(* Logix 5000 project; controller Project_Template vendor 1 type 14 code 106 rev 33.12; software revision 33.00 *)

TASK MainTask (continuous, watchdog 500 ms) : MainProgram

MODULES
   Local : vendor 1 type 14 code 106 (Compact 0, rev 33.12)
      Discrete_In_Slot_3 : 1769-IQ16 (Compact 3, rev 1.1, Input RPI 20 ms)
      Discrete_In_Slot_2 : 1769-IQ16 (Compact 2, rev 1.1, Input RPI 20 ms)
      ASCII_Slot_1 : vendor 1 type 109 code 66 (Compact 1, rev 2.1, Output RPI 100 ms)
      Discrete_Out_Slot_4 : 1769-OW16 (Compact 4, rev 1.1, Output RPI 20 ms)
      Discrete_Out_Slot_5 : 1769-OW16 (Compact 5, rev 1.1, Output RPI 20 ms)
END_MODULES

VAR_GLOBAL   (* controller tags *)
   AT_HOME : BOOL := 1;   // Home position
   AUTO : BOOL;   // Set Auto Process
   Box_Fell : BOOL;
   FLASH_FAST : BOOL;
   Flash_Fast_Off : TIMER := (PRE := 250);
   Flash_Fast_On : TIMER := (PRE := 250, ACC := 161, EN := 1, TT := 1);
   FLASH_MEDIUM : BOOL := 1;
   Flash_Medium_Off : TIMER := (PRE := 500, ACC := 161, EN := 1, TT := 1);
   Flash_Medium_On : TIMER := (PRE := 500, ACC := 500, EN := 1, DN := 1);
   FLASH_SLOW : BOOL;   // Slow Flashing
   Flash_Slow_Off : TIMER := (PRE := 1000);
   Flash_Slow_On : TIMER := (PRE := 1000, ACC := 664, EN := 1, TT := 1);
   I_Auto_Mode_Selector : ALIAS FOR Local:2:I.Data.2;
   I_Barcode_Stop_Raised : ALIAS FOR Local:3:I.Data.1;
   I_Box_Ejector_Extended : ALIAS FOR Local:2:I.Data.4;
   I_Reject_Cyl_Lowered : ALIAS FOR Local:3:I.Data.2;
   I_Reset_PB : ALIAS FOR Local:2:I.Data.3;
   I_Start_PB : ALIAS FOR Local:2:I.Data.0;
   I_Stop_PB : ALIAS FOR Local:2:I.Data.1;
   I_Vacuum_Head_at_Conveyor : ALIAS FOR Local:3:I.Data.0;
   I_Vacuum_Head_at_Magazine : ALIAS FOR Local:2:I.Data.15;
   I_Vacuum_Head_Extended : ALIAS FOR Local:2:I.Data.14;
   I_Vacuum_Head_Lowered : ALIAS FOR Local:2:I.Data.10;
   I_Vacuum_Head_Raised : ALIAS FOR Local:2:I.Data.9;
   I_Vacuum_Head_Retracted : ALIAS FOR Local:2:I.Data.13;
   I_Vacuum_Head_Rotated_CCW : ALIAS FOR Local:2:I.Data.11;
   I_Vacuum_Head_Rotated_CW : ALIAS FOR Local:2:I.Data.12;
   I_Vacuum_Sensor_On : ALIAS FOR Local:3:I.Data.8;
   O_Amber_Tower_Ind : ALIAS FOR Local:5:O.Data.9;
   O_Barcode_Stop_Raise : ALIAS FOR Local:4:O.Data.14;
   O_Box_Eject : ALIAS FOR Local:4:O.Data.0;
   O_Conveyor_On : ALIAS FOR Local:5:O.Data.5;
   O_Green_Tower_Ind : ALIAS FOR Local:5:O.Data.8;
   O_Red_Tower_Ind : ALIAS FOR Local:5:O.Data.10;
   O_Reject_Cyl_Extend : ALIAS FOR Local:5:O.Data.0;
   O_Reject_Cyl_Lower : ALIAS FOR Local:4:O.Data.15;
   O_Vacuum_Head_Extend : ALIAS FOR Local:4:O.Data.8;
   O_Vacuum_Head_Lower : ALIAS FOR Local:4:O.Data.5;
   O_Vacuum_Head_Rotate_CCW : ALIAS FOR Local:4:O.Data.7;
   O_Vacuum_Head_Rotate_CW : ALIAS FOR Local:4:O.Data.6;
   O_Vacuum_Head_to_Conveyor : ALIAS FOR Local:4:O.Data.9;
   O_Vacuum_Head_to_Magazine : ALIAS FOR Local:4:O.Data.10;
   O_Vacuum_Off : ALIAS FOR Local:5:O.Data.2;
   O_Vacuum_On : ALIAS FOR Local:5:O.Data.1;
   Production_Step : DINT := 11;
   Raise_Vacuum : BOOL;
   Reset_Step : DINT := 512;
   Retract_Box_Ejector : BOOL;
   Retract_Vacuum : BOOL;
   Status_IN_PRODUCTION : BOOL;
   Status_RESETTING : BOOL;
   Timer_Barcode_Delay : TIMER := (PRE := 1000);
   Timer_Conveyor_Delay : TIMER := (PRE := 500);
   Timer_Conveyor_Reset : TIMER := (PRE := 900, ACC := 900, EN := 1, DN := 1);   // Timer Conveyor to clear boxes
   Timer_Extend_Delay : TIMER := (PRE := 2000, ACC := 296, EN := 1, TT := 1);
   Timer_Pre_Production : TIMER := (PRE := 500, ACC := 500, EN := 1, DN := 1);
   Timer_Pre_Reset : TIMER := (PRE := 500);
   Timer_Reset : TIMER[7] := ([0].PRE := 250, [1].PRE := 250, [2].PRE := 250, [3].PRE := 250, [4].PRE := 250, [5].PRE := 300, [6].PRE := 125);
   Timer_Vacuum_Delay : TIMER := (PRE := 250, ACC := 250, EN := 1, DN := 1);
END_VAR

PROGRAM MainProgram   (* main routine MainRoutine *)

ROUTINE a_Reset_Routine   (* ladder *)
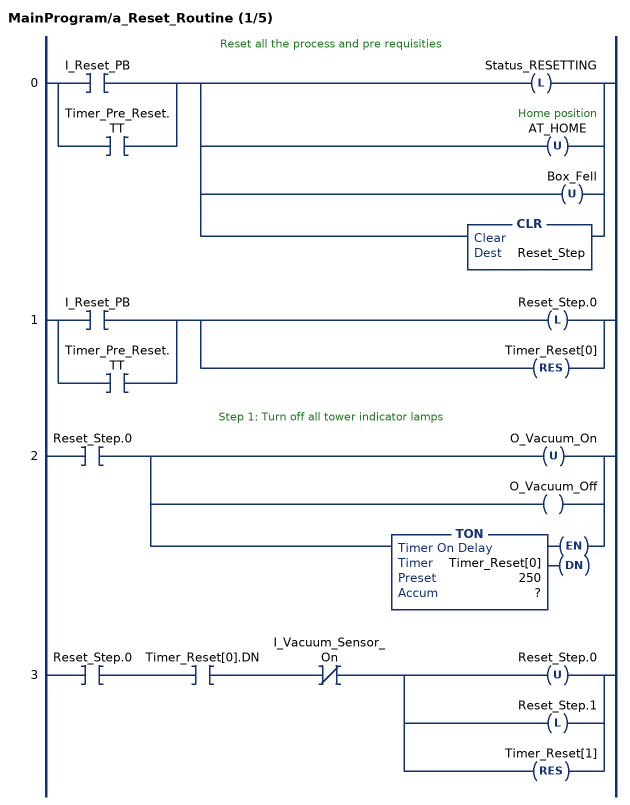
   // Reset all the process and pre requisities
   0: [XIC(I_Reset_PB) ,XIC(Timer_Pre_Reset.TT) ][OTL(Status_RESETTING) ,OTU(AT_HOME) ,OTU(Box_Fell) ,CLR(Reset_Step) ];
   1: [XIC(I_Reset_PB) ,XIC(Timer_Pre_Reset.TT) ][OTL(Reset_Step.0) ,RES(Timer_Reset[0]) ];
   // Step 1: Turn off all tower indicator lamps
   2: XIC(Reset_Step.0)[OTU(O_Vacuum_On) ,OTE(O_Vacuum_Off) ,TON(Timer_Reset[0],?,?) ];
   3: XIC(Reset_Step.0)XIC(Timer_Reset[0].DN)XIO(I_Vacuum_Sensor_On)[OTU(Reset_Step.0) ,OTL(Reset_Step.1) ,RES(Timer_Reset[1]) ];
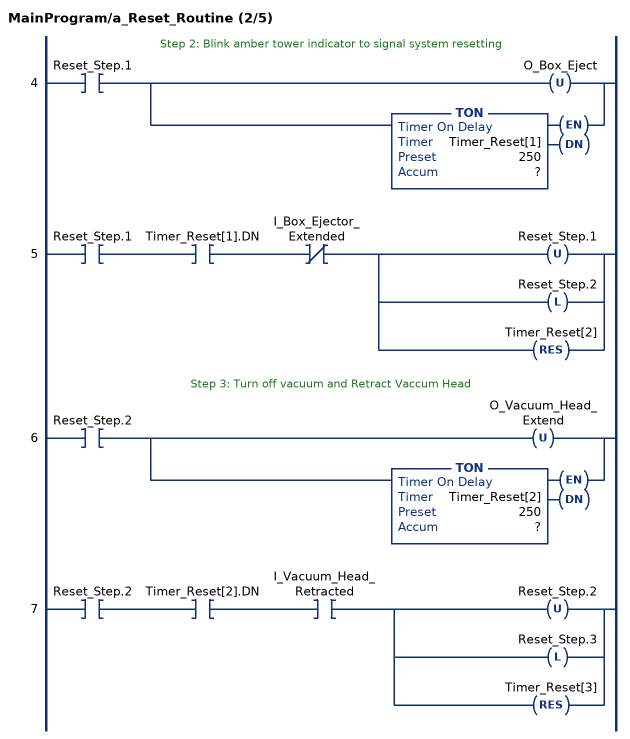
   // Step 2: Blink amber tower indicator to signal system resetting
   4: XIC(Reset_Step.1)[OTU(O_Box_Eject) ,TON(Timer_Reset[1],?,?) ];
   5: XIC(Reset_Step.1)XIC(Timer_Reset[1].DN)XIO(I_Box_Ejector_Extended)[OTU(Reset_Step.1) ,OTL(Reset_Step.2) ,RES(Timer_Reset[2]) ];
   // Step 3: Turn off vacuum and Retract Vaccum Head
   6: XIC(Reset_Step.2)[OTU(O_Vacuum_Head_Extend) ,TON(Timer_Reset[2],?,?) ];
   7: XIC(Reset_Step.2)XIC(Timer_Reset[2].DN)XIC(I_Vacuum_Head_Retracted)[OTU(Reset_Step.2) ,OTL(Reset_Step.3) ,RES(Timer_Reset[3]) ];
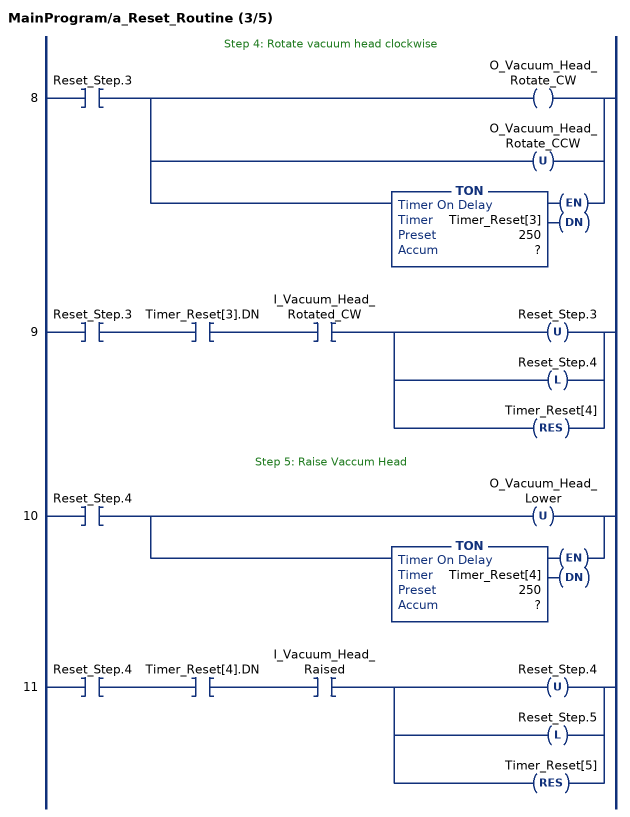
   // Step 4: Rotate vacuum head clockwise
   8: XIC(Reset_Step.3)[OTE(O_Vacuum_Head_Rotate_CW) ,OTU(O_Vacuum_Head_Rotate_CCW) ,TON(Timer_Reset[3],?,?) ];
   9: XIC(Reset_Step.3)XIC(Timer_Reset[3].DN)XIC(I_Vacuum_Head_Rotated_CW)[OTU(Reset_Step.3) ,OTL(Reset_Step.4) ,RES(Timer_Reset[4]) ];
   // Step 5: Raise Vaccum Head
   10: XIC(Reset_Step.4)[OTU(O_Vacuum_Head_Lower) ,TON(Timer_Reset[4],?,?) ];
   11: XIC(Reset_Step.4)XIC(Timer_Reset[4].DN)XIC(I_Vacuum_Head_Raised)[OTU(Reset_Step.4) ,OTL(Reset_Step.5) ,RES(Timer_Reset[5]) ];
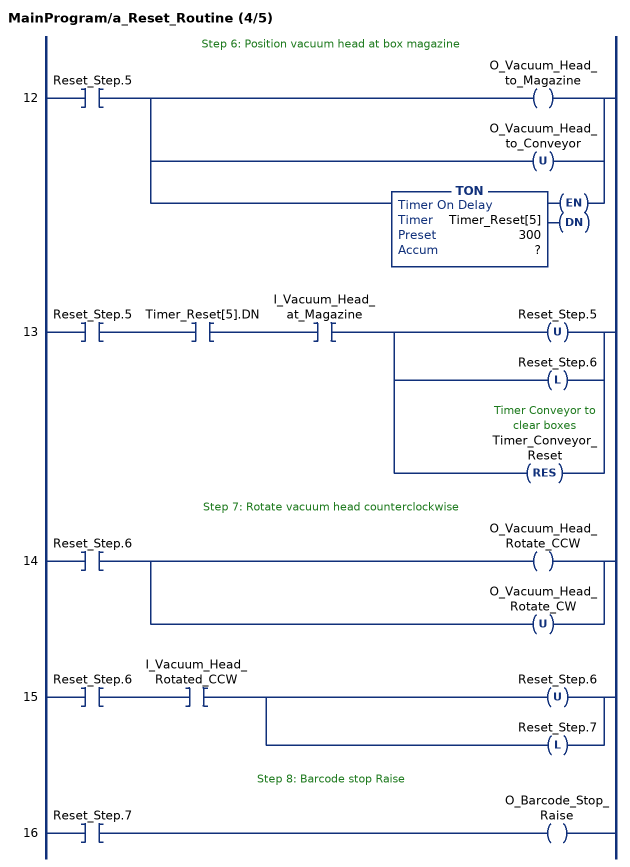
   // Step 6: Position vacuum head at box magazine
   12: XIC(Reset_Step.5)[OTE(O_Vacuum_Head_to_Magazine) ,OTU(O_Vacuum_Head_to_Conveyor) ,TON(Timer_Reset[5],?,?) ];
   13: XIC(Reset_Step.5)XIC(Timer_Reset[5].DN)XIC(I_Vacuum_Head_at_Magazine)[OTU(Reset_Step.5) ,OTL(Reset_Step.6) ,RES(Timer_Conveyor_Reset) ];
   // Step 7: Rotate vacuum head counterclockwise
   14: XIC(Reset_Step.6)[OTE(O_Vacuum_Head_Rotate_CCW) ,OTU(O_Vacuum_Head_Rotate_CW) ];
   15: XIC(Reset_Step.6)XIC(I_Vacuum_Head_Rotated_CCW)[OTU(Reset_Step.6) ,OTL(Reset_Step.7) ];
   // Step 8: Barcode stop Raise
   16: XIC(Reset_Step.7)OTE(O_Barcode_Stop_Raise);
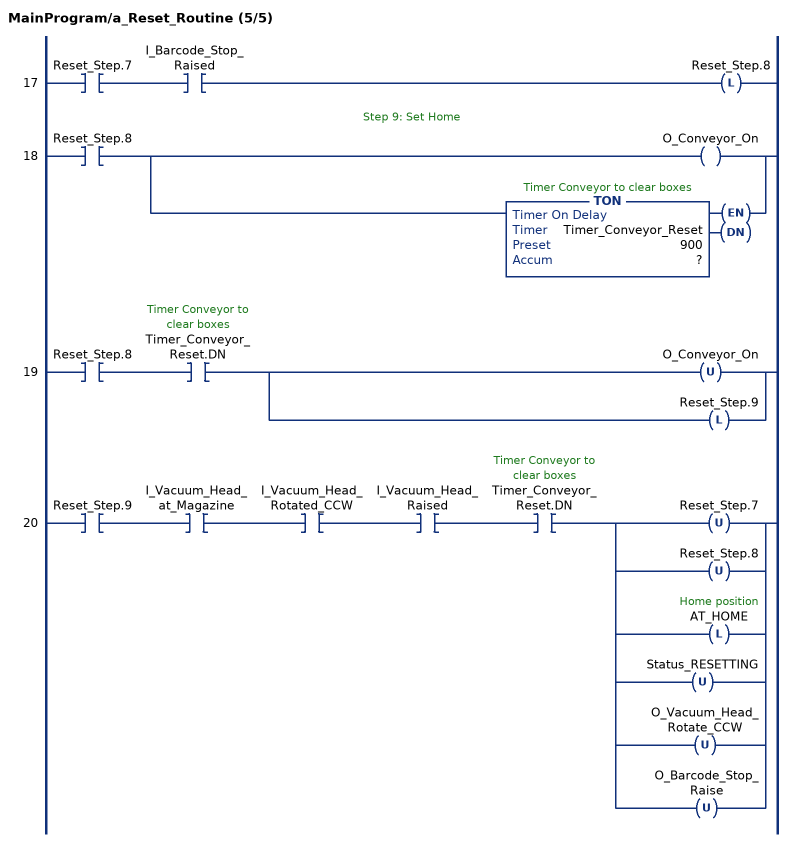
   17: XIC(Reset_Step.7)XIC(I_Barcode_Stop_Raised)OTL(Reset_Step.8);
   // Step 9: Set Home
   18: XIC(Reset_Step.8)[OTE(O_Conveyor_On) ,TON(Timer_Conveyor_Reset,?,?) ];
   19: XIC(Reset_Step.8)XIC(Timer_Conveyor_Reset.DN)[OTU(O_Conveyor_On) ,OTL(Reset_Step.9) ];
   20: XIC(Reset_Step.9)XIC(I_Vacuum_Head_at_Magazine)XIC(I_Vacuum_Head_Rotated_CCW)XIC(I_Vacuum_Head_Raised)XIC(Timer_Conveyor_Reset.DN)[OTU(Reset_Step.7) ,OTU(Reset_Step.8) ,OTL(AT_HOME) ,OTU(Status_RESETTING) ,OTU(O_Vacuum_Head_Rotate_CCW) ,OTU(O_Barcode_Stop_Raise) ];
END_ROUTINE

ROUTINE b_Production_Routine   (* ladder *)
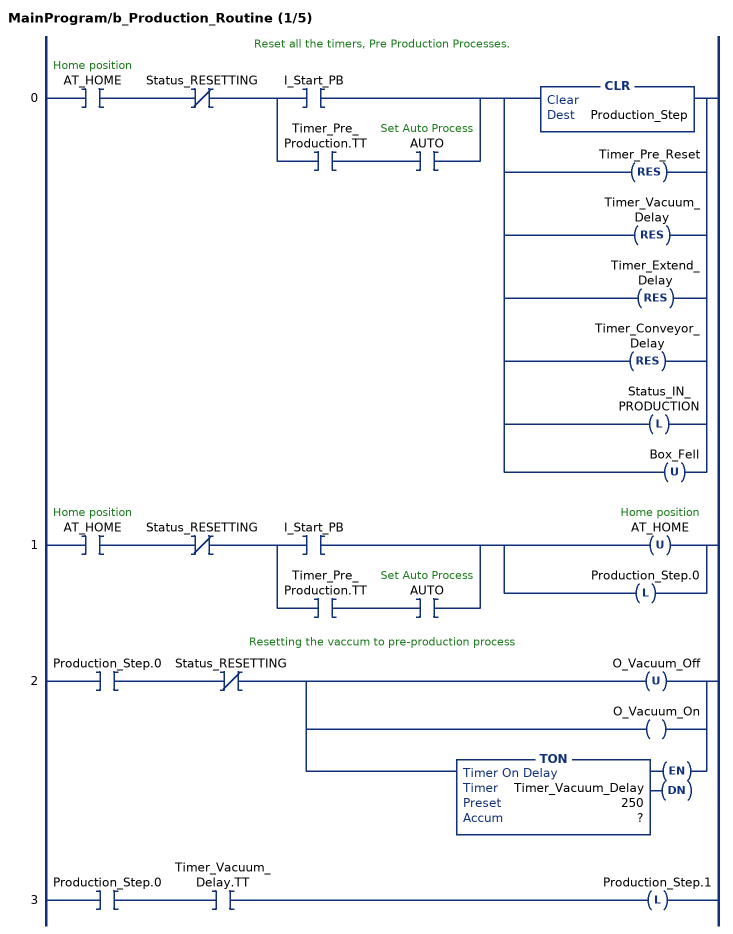
   // Reset all the timers, Pre Production Processes.
   0: XIC(AT_HOME)XIO(Status_RESETTING)[XIC(I_Start_PB) ,XIC(Timer_Pre_Production.TT) XIC(AUTO) ][CLR(Production_Step) ,RES(Timer_Pre_Reset) ,RES(Timer_Vacuum_Delay) ,RES(Timer_Extend_Delay) ,RES(Timer_Conveyor_Delay) ,OTL(Status_IN_PRODUCTION) ,OTU(Box_Fell) ];
   1: XIC(AT_HOME)XIO(Status_RESETTING)[XIC(I_Start_PB) ,XIC(Timer_Pre_Production.TT) XIC(AUTO) ][OTU(AT_HOME) ,OTL(Production_Step.0) ];
   // Resetting the vaccum to pre-production process
   2: XIC(Production_Step.0)XIO(Status_RESETTING)[OTU(O_Vacuum_Off) ,OTE(O_Vacuum_On) ,TON(Timer_Vacuum_Delay,?,?) ];
   3: XIC(Production_Step.0)XIC(Timer_Vacuum_Delay.TT)OTL(Production_Step.1);
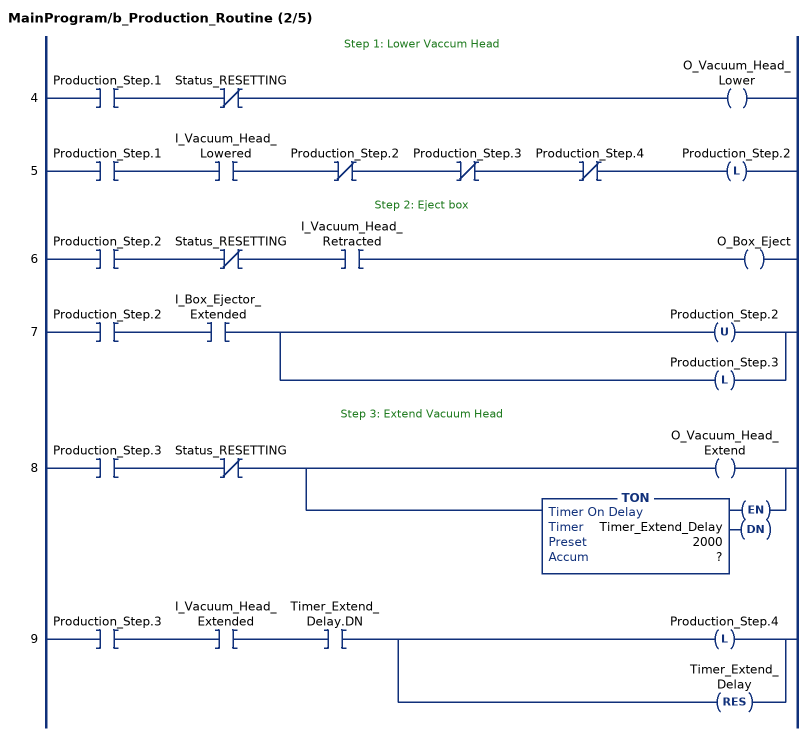
   // Step 1: Lower Vaccum Head
   4: XIC(Production_Step.1)XIO(Status_RESETTING)OTE(O_Vacuum_Head_Lower);
   5: XIC(Production_Step.1)XIC(I_Vacuum_Head_Lowered)XIO(Production_Step.2)XIO(Production_Step.3)XIO(Production_Step.4)OTL(Production_Step.2);
   // Step 2: Eject box
   6: XIC(Production_Step.2)XIO(Status_RESETTING)XIC(I_Vacuum_Head_Retracted)OTE(O_Box_Eject);
   7: XIC(Production_Step.2)XIC(I_Box_Ejector_Extended)[OTU(Production_Step.2) ,OTL(Production_Step.3) ];
   // Step 3: Extend Vacuum Head
   8: XIC(Production_Step.3)XIO(Status_RESETTING)[OTE(O_Vacuum_Head_Extend) ,TON(Timer_Extend_Delay,?,?) ];
   9: XIC(Production_Step.3)XIC(I_Vacuum_Head_Extended)XIC(Timer_Extend_Delay.DN)[OTL(Production_Step.4) ,RES(Timer_Extend_Delay) ];
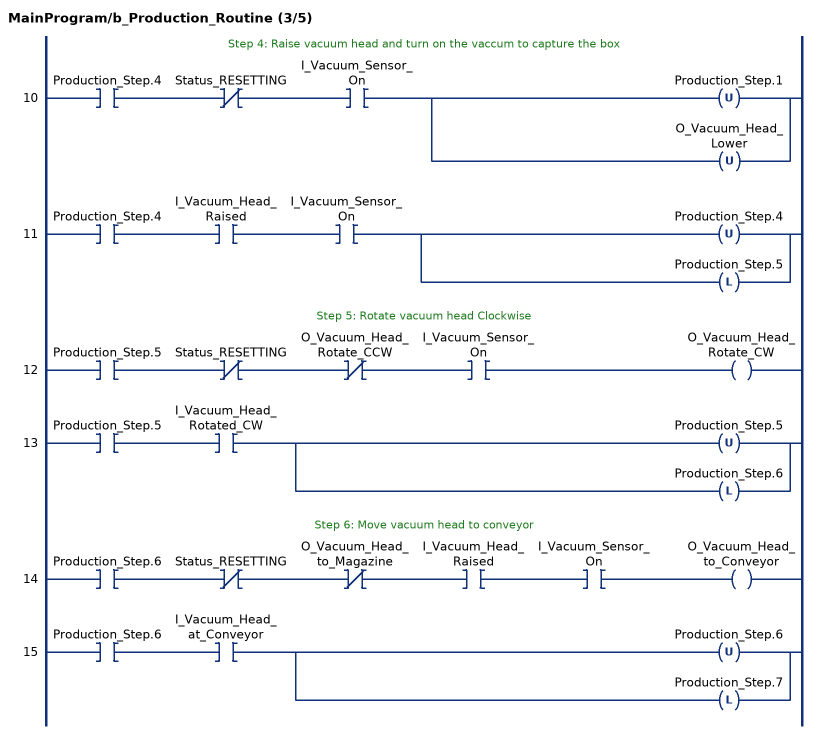
   // Step 4: Raise vacuum head and turn on the vaccum to capture the box
   10: XIC(Production_Step.4)XIO(Status_RESETTING)XIC(I_Vacuum_Sensor_On)[OTU(Production_Step.1) ,OTU(O_Vacuum_Head_Lower) ];
   11: XIC(Production_Step.4)XIC(I_Vacuum_Head_Raised)XIC(I_Vacuum_Sensor_On)[OTU(Production_Step.4) ,OTL(Production_Step.5) ];
   // Step 5: Rotate vacuum head Clockwise
   12: XIC(Production_Step.5)XIO(Status_RESETTING)XIO(O_Vacuum_Head_Rotate_CCW)XIC(I_Vacuum_Sensor_On)OTE(O_Vacuum_Head_Rotate_CW);
   13: XIC(Production_Step.5)XIC(I_Vacuum_Head_Rotated_CW)[OTU(Production_Step.5) ,OTL(Production_Step.6) ];
   // Step 6: Move vacuum head to conveyor
   14: XIC(Production_Step.6)XIO(Status_RESETTING)XIO(O_Vacuum_Head_to_Magazine)XIC(I_Vacuum_Head_Raised)XIC(I_Vacuum_Sensor_On)OTE(O_Vacuum_Head_to_Conveyor);
   15: XIC(Production_Step.6)XIC(I_Vacuum_Head_at_Conveyor)[OTU(Production_Step.6) ,OTL(Production_Step.7) ];
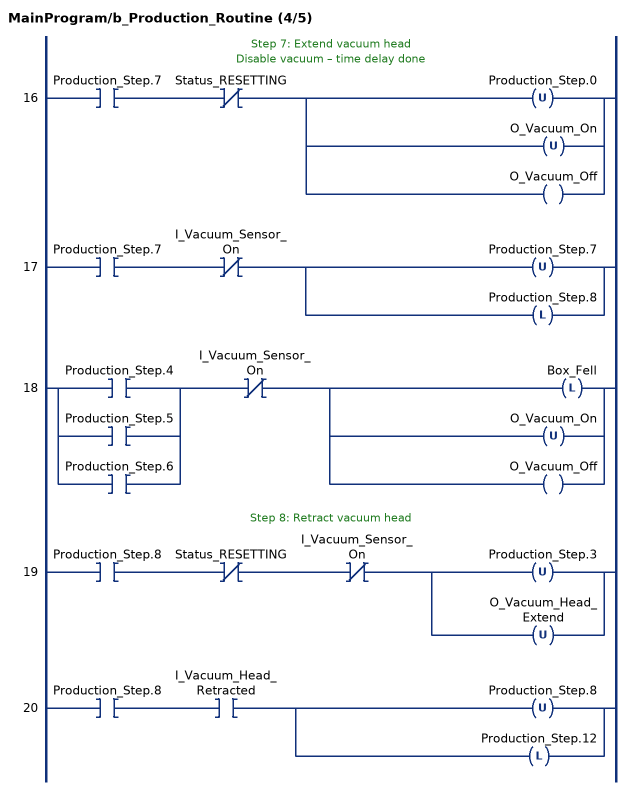
   // Step 7: Extend vacuum head
   // Disable vacuum – time delay done
   16: XIC(Production_Step.7)XIO(Status_RESETTING)[OTU(Production_Step.0) ,OTU(O_Vacuum_On) ,OTE(O_Vacuum_Off) ];
   17: XIC(Production_Step.7)XIO(I_Vacuum_Sensor_On)[OTU(Production_Step.7) ,OTL(Production_Step.8) ];
   18: [XIC(Production_Step.4) ,XIC(Production_Step.5) ,XIC(Production_Step.6) ]XIO(I_Vacuum_Sensor_On)[OTL(Box_Fell) ,OTU(O_Vacuum_On) ,OTE(O_Vacuum_Off) ];
   // Step 8: Retract vacuum head
   19: XIC(Production_Step.8)XIO(Status_RESETTING)XIO(I_Vacuum_Sensor_On)[OTU(Production_Step.3) ,OTU(O_Vacuum_Head_Extend) ];
   20: XIC(Production_Step.8)XIC(I_Vacuum_Head_Retracted)[OTU(Production_Step.8) ,OTL(Production_Step.12) ];
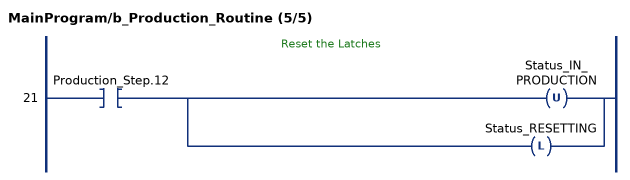
   // Reset the Latches
   21: XIC(Production_Step.12)[OTU(Status_IN_PRODUCTION) ,OTL(Status_RESETTING) ];
END_ROUTINE

ROUTINE c_AutoProcess_Routine   (* ladder *)
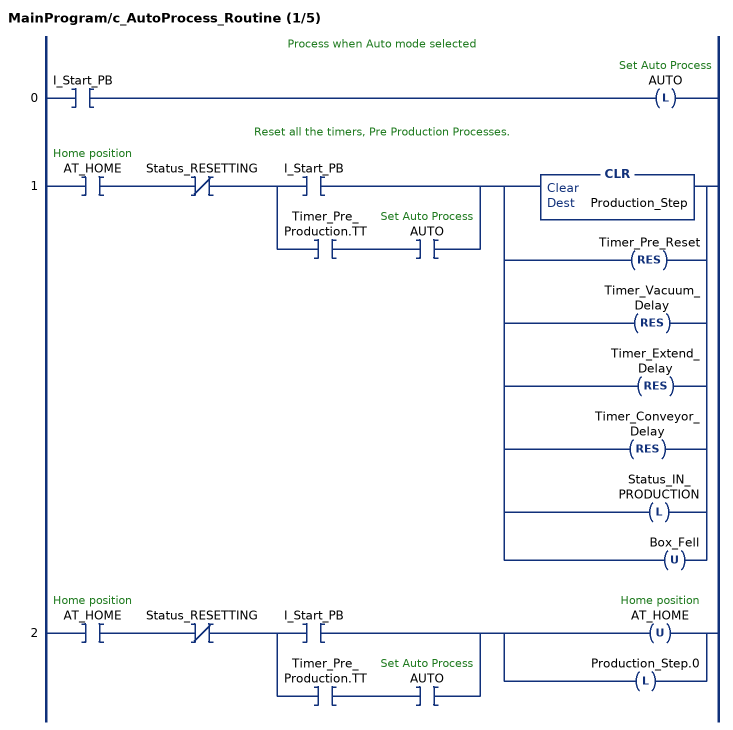
   // Process when Auto mode selected
   0: XIC(I_Start_PB)OTL(AUTO);
   // Reset all the timers, Pre Production Processes.
   1: XIC(AT_HOME)XIO(Status_RESETTING)[XIC(I_Start_PB) ,XIC(Timer_Pre_Production.TT) XIC(AUTO) ][CLR(Production_Step) ,RES(Timer_Pre_Reset) ,RES(Timer_Vacuum_Delay) ,RES(Timer_Extend_Delay) ,RES(Timer_Conveyor_Delay) ,OTL(Status_IN_PRODUCTION) ,OTU(Box_Fell) ];
   2: XIC(AT_HOME)XIO(Status_RESETTING)[XIC(I_Start_PB) ,XIC(Timer_Pre_Production.TT) XIC(AUTO) ][OTU(AT_HOME) ,OTL(Production_Step.0) ];
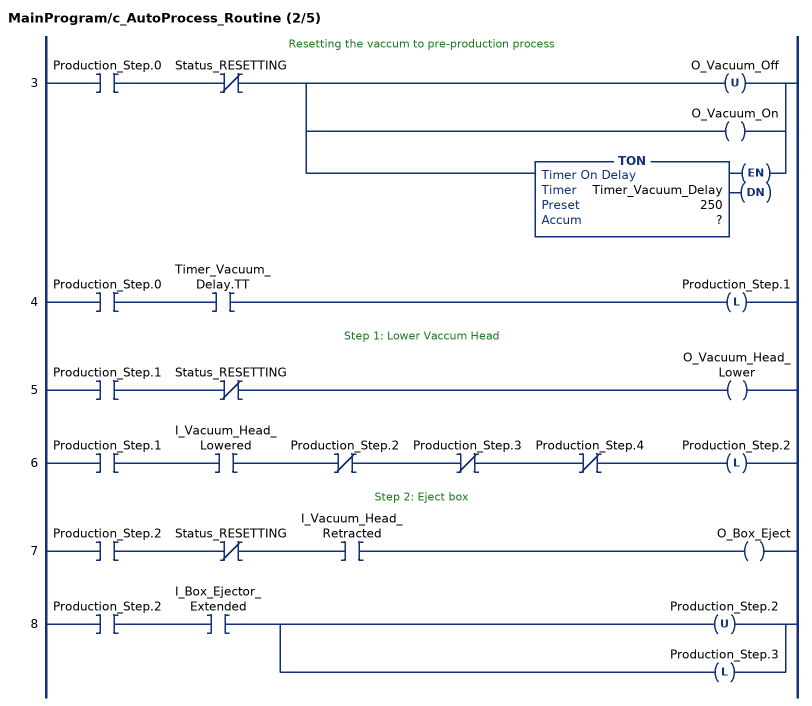
   // Resetting the vaccum to pre-production process
   3: XIC(Production_Step.0)XIO(Status_RESETTING)[OTU(O_Vacuum_Off) ,OTE(O_Vacuum_On) ,TON(Timer_Vacuum_Delay,?,?) ];
   4: XIC(Production_Step.0)XIC(Timer_Vacuum_Delay.TT)OTL(Production_Step.1);
   // Step 1: Lower Vaccum Head
   5: XIC(Production_Step.1)XIO(Status_RESETTING)OTE(O_Vacuum_Head_Lower);
   6: XIC(Production_Step.1)XIC(I_Vacuum_Head_Lowered)XIO(Production_Step.2)XIO(Production_Step.3)XIO(Production_Step.4)OTL(Production_Step.2);
   // Step 2: Eject box
   7: XIC(Production_Step.2)XIO(Status_RESETTING)XIC(I_Vacuum_Head_Retracted)OTE(O_Box_Eject);
   8: XIC(Production_Step.2)XIC(I_Box_Ejector_Extended)[OTU(Production_Step.2) ,OTL(Production_Step.3) ];
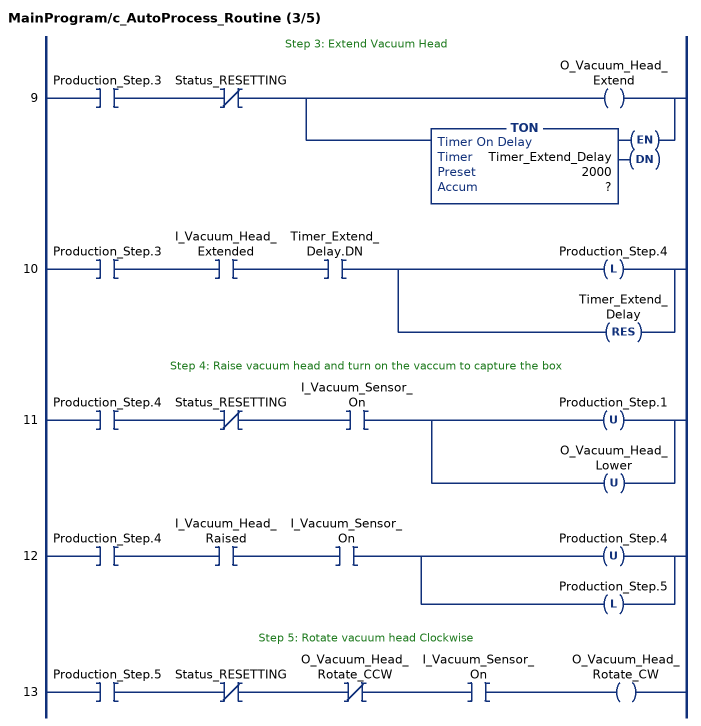
   // Step 3: Extend Vacuum Head
   9: XIC(Production_Step.3)XIO(Status_RESETTING)[OTE(O_Vacuum_Head_Extend) ,TON(Timer_Extend_Delay,?,?) ];
   10: XIC(Production_Step.3)XIC(I_Vacuum_Head_Extended)XIC(Timer_Extend_Delay.DN)[OTL(Production_Step.4) ,RES(Timer_Extend_Delay) ];
   // Step 4: Raise vacuum head and turn on the vaccum to capture the box
   11: XIC(Production_Step.4)XIO(Status_RESETTING)XIC(I_Vacuum_Sensor_On)[OTU(Production_Step.1) ,OTU(O_Vacuum_Head_Lower) ];
   12: XIC(Production_Step.4)XIC(I_Vacuum_Head_Raised)XIC(I_Vacuum_Sensor_On)[OTU(Production_Step.4) ,OTL(Production_Step.5) ];
   // Step 5: Rotate vacuum head Clockwise
   13: XIC(Production_Step.5)XIO(Status_RESETTING)XIO(O_Vacuum_Head_Rotate_CCW)XIC(I_Vacuum_Sensor_On)OTE(O_Vacuum_Head_Rotate_CW);
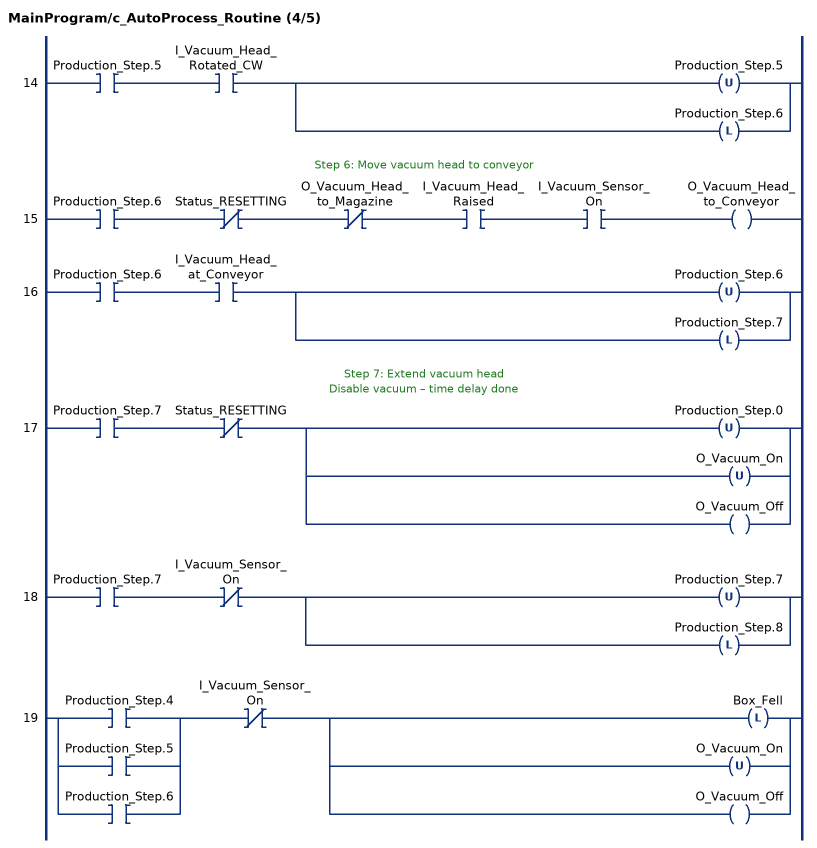
   14: XIC(Production_Step.5)XIC(I_Vacuum_Head_Rotated_CW)[OTU(Production_Step.5) ,OTL(Production_Step.6) ];
   // Step 6: Move vacuum head to conveyor
   15: XIC(Production_Step.6)XIO(Status_RESETTING)XIO(O_Vacuum_Head_to_Magazine)XIC(I_Vacuum_Head_Raised)XIC(I_Vacuum_Sensor_On)OTE(O_Vacuum_Head_to_Conveyor);
   16: XIC(Production_Step.6)XIC(I_Vacuum_Head_at_Conveyor)[OTU(Production_Step.6) ,OTL(Production_Step.7) ];
   // Step 7: Extend vacuum head
   // Disable vacuum – time delay done
   17: XIC(Production_Step.7)XIO(Status_RESETTING)[OTU(Production_Step.0) ,OTU(O_Vacuum_On) ,OTE(O_Vacuum_Off) ];
   18: XIC(Production_Step.7)XIO(I_Vacuum_Sensor_On)[OTU(Production_Step.7) ,OTL(Production_Step.8) ];
   19: [XIC(Production_Step.4) ,XIC(Production_Step.5) ,XIC(Production_Step.6) ]XIO(I_Vacuum_Sensor_On)[OTL(Box_Fell) ,OTU(O_Vacuum_On) ,OTE(O_Vacuum_Off) ];
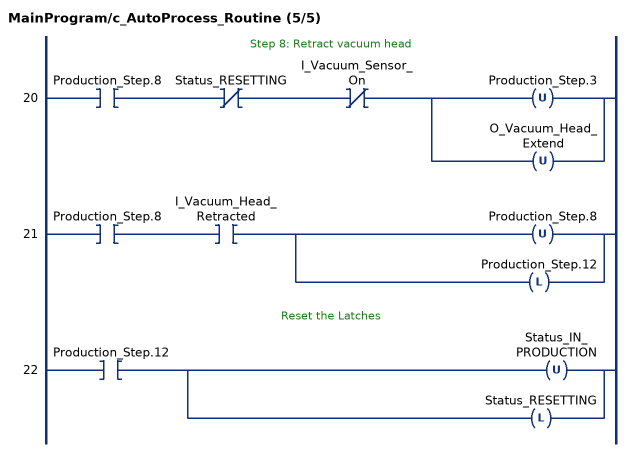
   // Step 8: Retract vacuum head
   20: XIC(Production_Step.8)XIO(Status_RESETTING)XIO(I_Vacuum_Sensor_On)[OTU(Production_Step.3) ,OTU(O_Vacuum_Head_Extend) ];
   21: XIC(Production_Step.8)XIC(I_Vacuum_Head_Retracted)[OTU(Production_Step.8) ,OTL(Production_Step.12) ];
   // Reset the Latches
   22: XIC(Production_Step.12)[OTU(Status_IN_PRODUCTION) ,OTL(Status_RESETTING) ];
END_ROUTINE

ROUTINE MainRoutine   (* ladder *)
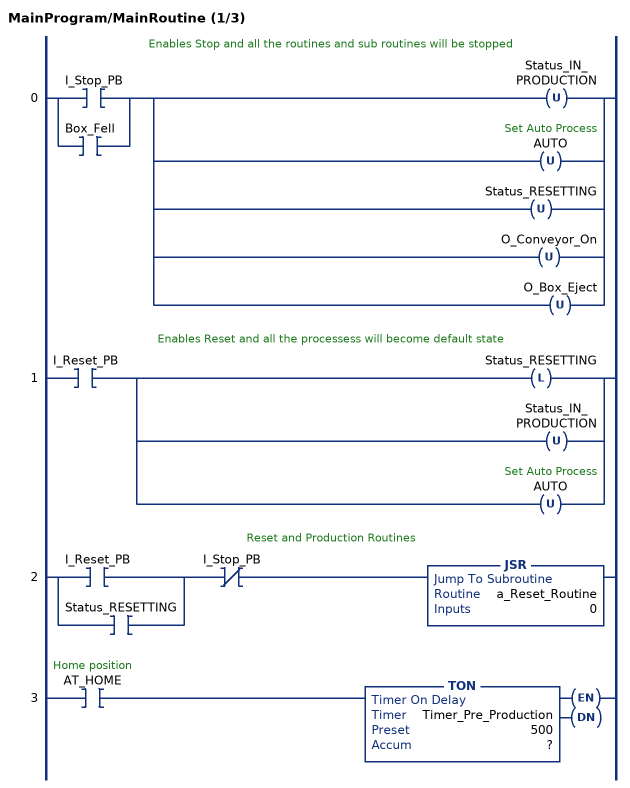
   // Enables Stop and all the routines and sub routines will be stopped
   0: [XIC(I_Stop_PB) ,XIC(Box_Fell) ][OTU(Status_IN_PRODUCTION) ,OTU(AUTO) ,OTU(Status_RESETTING) ,OTU(O_Conveyor_On) ,OTU(O_Box_Eject) ];
   // Enables Reset and all the processess will become default state
   1: XIC(I_Reset_PB)[OTL(Status_RESETTING) ,OTU(Status_IN_PRODUCTION) ,OTU(AUTO) ];
   // Reset and Production Routines
   2: [XIC(I_Reset_PB) ,XIC(Status_RESETTING) ]XIO(I_Stop_PB)JSR(a_Reset_Routine,0);
   3: XIC(AT_HOME)TON(Timer_Pre_Production,?,?);
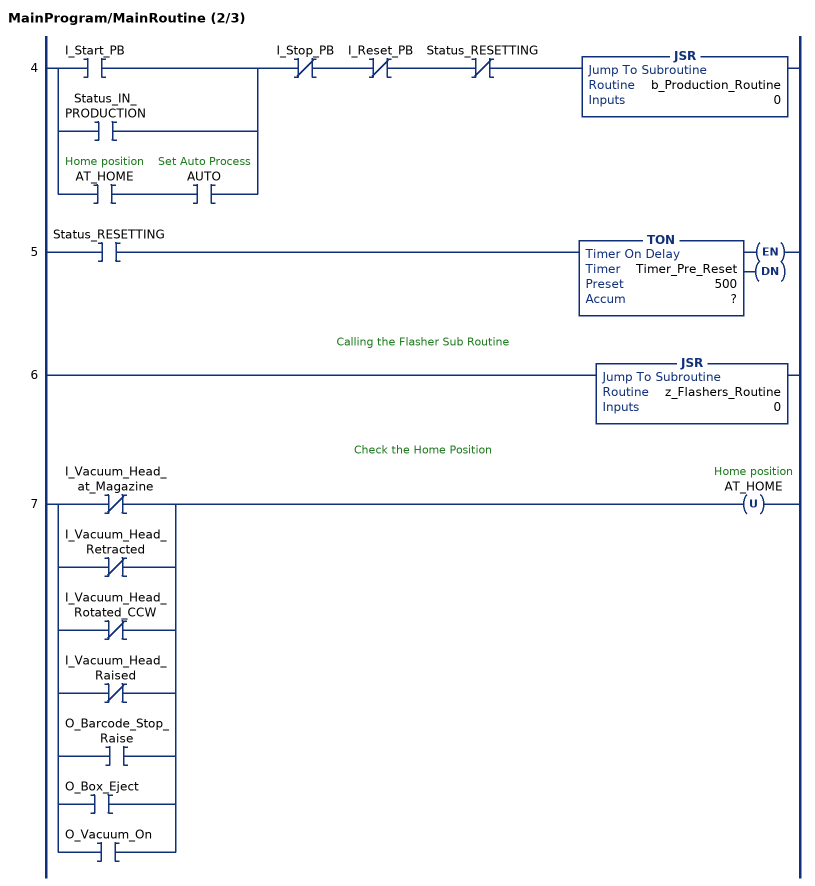
   4: [XIC(I_Start_PB) ,XIC(Status_IN_PRODUCTION) ,XIC(AT_HOME) XIC(AUTO) ]XIO(I_Stop_PB)XIO(I_Reset_PB)XIO(Status_RESETTING)JSR(b_Production_Routine,0);
   5: XIC(Status_RESETTING)TON(Timer_Pre_Reset,?,?);
   // Calling the Flasher Sub Routine
   6: JSR(z_Flashers_Routine,0);
   // Check the Home Position
   7: [XIO(I_Vacuum_Head_at_Magazine) ,XIO(I_Vacuum_Head_Retracted) ,XIO(I_Vacuum_Head_Rotated_CCW) ,XIO(I_Vacuum_Head_Raised) ,XIC(O_Barcode_Stop_Raise) ,XIC(O_Box_Eject) ,XIC(O_Vacuum_On) ]OTU(AT_HOME);
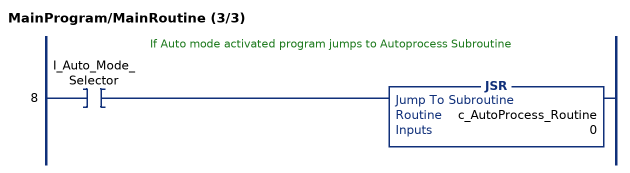
   // If Auto mode activated program jumps to Autoprocess Subroutine
   8: XIC(I_Auto_Mode_Selector)JSR(c_AutoProcess_Routine,0);
END_ROUTINE

ROUTINE z_Flashers_Routine   (* ladder *)
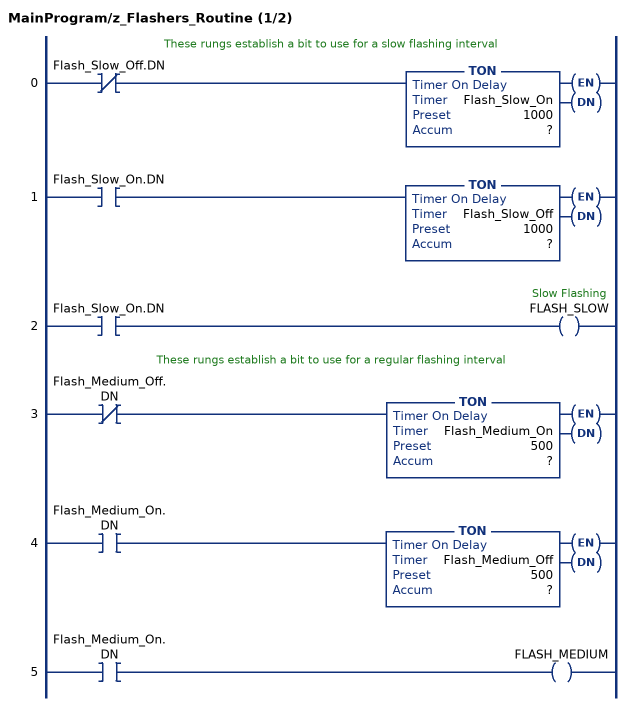
   // These rungs establish a bit to use for a slow flashing interval
   0: XIO(Flash_Slow_Off.DN)TON(Flash_Slow_On,?,?);
   1: XIC(Flash_Slow_On.DN)TON(Flash_Slow_Off,?,?);
   2: XIC(Flash_Slow_On.DN)OTE(FLASH_SLOW);
   // These rungs establish a bit to use for a regular flashing interval
   3: XIO(Flash_Medium_Off.DN)TON(Flash_Medium_On,?,?);
   4: XIC(Flash_Medium_On.DN)TON(Flash_Medium_Off,?,?);
   5: XIC(Flash_Medium_On.DN)OTE(FLASH_MEDIUM);
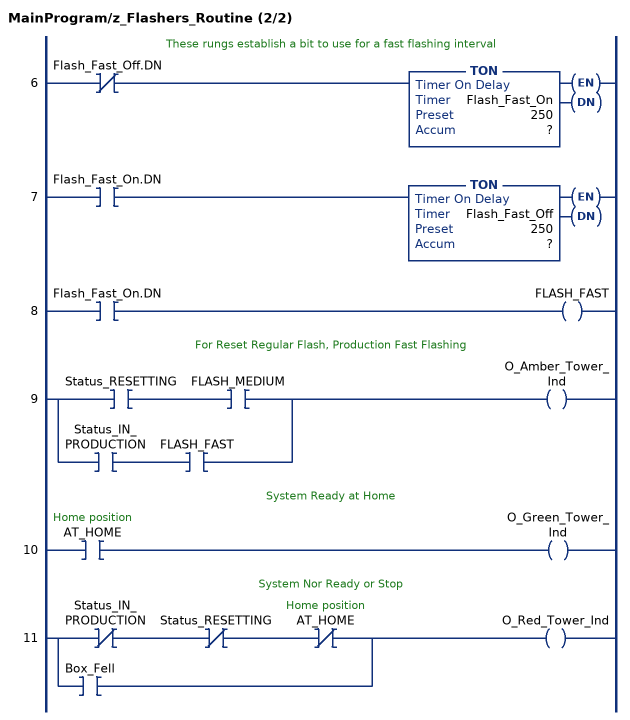
   // These rungs establish a bit to use for a fast flashing interval
   6: XIO(Flash_Fast_Off.DN)TON(Flash_Fast_On,?,?);
   7: XIC(Flash_Fast_On.DN)TON(Flash_Fast_Off,?,?);
   8: XIC(Flash_Fast_On.DN)OTE(FLASH_FAST);
   // For Reset Regular Flash, Production Fast Flashing
   9: [XIC(Status_RESETTING) XIC(FLASH_MEDIUM) ,XIC(Status_IN_PRODUCTION) XIC(FLASH_FAST) ]OTE(O_Amber_Tower_Ind);
   // System Ready at Home
   10: XIC(AT_HOME)OTE(O_Green_Tower_Ind);
   // System Nor Ready or Stop
   11: [XIO(Status_IN_PRODUCTION) XIO(Status_RESETTING) XIO(AT_HOME) ,XIC(Box_Fell) ]OTE(O_Red_Tower_Ind);
END_ROUTINE
END_PROGRAM
